INTERFACE I_Stack EXTENDS I_Collection

// Gets an immutable list of the items in the stack.
PROPERTY _Values : I_Immutable_List
GET
END_GET
END_PROPERTY

// Empties/Clears/Deletes every item in the stack.
METHOD Clear : I_Stack
END_METHOD

// Gets item at the top of the stack.
METHOD Get : I_Stack
VAR_INPUT
	Item : ANY; // Variable to store returned item value. 
END_VAR
VAR_OUTPUT
	bSuccess : BOOL;
END_VAR
END_METHOD

// Gets item at the top of the stack as a generic.
METHOD Get_Generic : I_Stack
VAR_OUTPUT
	Item : T_Generic; // Variable to store returned item value
	bSuccess : BOOL;
END_VAR
END_METHOD

// Removes item at the top of the stack without returning anything.
METHOD Pop : I_Stack
VAR_OUTPUT
	bSuccess : BOOL;
END_VAR
END_METHOD

// Add item to the top of the stack.
METHOD Push : I_Stack
VAR_INPUT
	Item : ANY; // Item to store.
END_VAR
VAR_OUTPUT
	bSuccess : BOOL;
END_VAR
END_METHOD

// Add generic item to the top of the stack.
METHOD Push_Generic : I_Stack
VAR_INPUT
	Item : T_Generic; // Item to store.
END_VAR
VAR_OUTPUT
	bSuccess : BOOL;
END_VAR
END_METHOD

// Reverses order of items on stack.
METHOD Reverse : I_Stack
VAR_OUTPUT
	bSuccess : BOOL;
END_VAR
END_METHOD

END_INTERFACE

(* stored: Version 1.1.0.1
   Itf I_Stack: Id {154dbc22-ff0e-03ac-018a-f60dfa7fd15f}
   Property _Values: Id {29199d50-f613-0bc4-2c63-f9fe06b9c482}
   Get Get: Id {ca8fc136-58b9-020d-3adb-f1df59ebe1ed}
   Method Clear: Id {1373b957-329a-0b05-0b47-3978fc3bd5a2}
   Method Get: Id {60584d29-80a2-0f00-3f32-146bf021e1d4}
   Method Get_Generic: Id {1f7362cc-4b55-06a3-2809-ad8ef9d7f2c5}
   Method Pop: Id {e7f906f2-44e7-0e51-1e35-4f1700cbc6c0}
   Method Push: Id {0cb19a43-3d3b-0071-25c7-aaddce41cb24}
   Method Push_Generic: Id {4d82994d-305a-0f32-0bbe-c3540dc33ada}
   Method Reverse: Id {2b820956-17bb-0a3b-0a83-dc66d5beef77} *)
